{attribute addProperty BoxType "KL3351-0003"}
{attribute addProperty Id "Channel_1Channel_83E614FE00"}
{attribute addProperty CRC "4023379778"}
{attribute addProperty SizeInBites "0"}
{attribute addProperty SizeInBytes "0"}
TYPE KL_EFCFE742 :
STRUCT
	{attribute addProperty Name "Channel_1"}
	Channel_1 : Channel_83E614FE;
END_STRUCT
END_TYPE

(* stored: Version 1.2.0.0, ProductVersion 3.1.4024.9
   DUT KL_EFCFE742: Id {199631b1-5c65-4966-8f04-67e548d66bd0} *)
